// TIA Portal V20 export
TYPE "IOInterface"
   STRUCT
      DI_001 : "IO_DI";
      DO_001 : "IO_DO";
      AI_001 : "IO_AI";
      AO_001 : "IO_AO";
      VSD_001 { ExternalAccessible := 'False'; ExternalVisible := 'False'; ExternalWritable := 'False'} : "IO_VSD";
      MOT_001 { ExternalAccessible := 'False'; ExternalVisible := 'False'; ExternalWritable := 'False'} : "IO_MOT";
      VLV_001 { ExternalAccessible := 'False'; ExternalVisible := 'False'; ExternalWritable := 'False'} : "IO_VLV";
      CONTVLV_001 { ExternalAccessible := 'False'; ExternalVisible := 'False'; ExternalWritable := 'False'} : "IO_CONTVLV";
   END_STRUCT;
END_TYPE
